// TIA Portal V17 export
// export: Created 2023-05-07T12:08:10.5778638Z, ExportSetting WithDefaults, DisplayName Totally Integrated Automation Portal, DisplayVersion V17, DisplayName TIA Portal Openness, DisplayVersion V17, DisplayName TIA Portal Version Control Interface, DisplayVersion V17, DisplayName TIA Portal Test Suite Advanced, DisplayVersion V17, DisplayName STEP 7 Professional, DisplayVersion V17, DisplayName SIMATIC Energy Suite, DisplayVersion V17, DisplayName STEP 7 Safety, DisplayVersion V17, DisplayName WinCC Professional, DisplayVersion V17
ORGANIZATION_BLOCK "Main"   // OB1, LAD, ProgramCycle
TITLE = "Main Program Sweep (Cycle)"
{ S7_Optimized_Access := 'TRUE' }
VERSION : 0.1
// stored: AutoNumber true, IsIECCheckEnabled false, SetENOAutomatically false
   VAR_INPUT
      Initial_Call : Bool;   // Initial call of this OB
      Remanence : Bool;   // =True, if remanent data are available
   END_VAR
BEGIN

REGION Network 1: Call: MHJ-PLC-Lab-Function-S71500
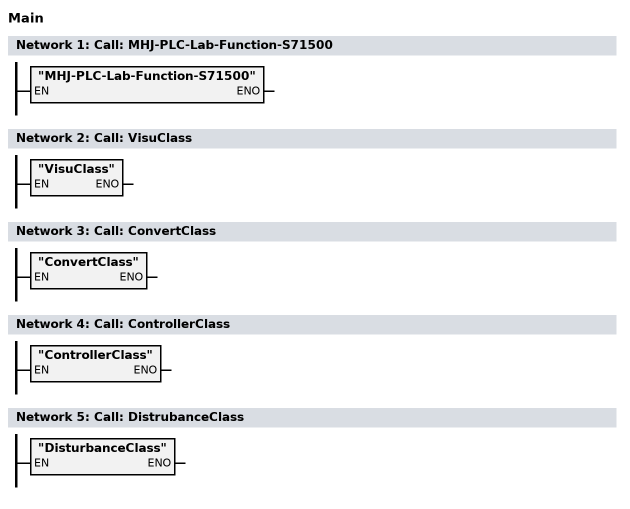
   RUNG wire#powerrail
      "MHJ-PLC-Lab-Function-S71500"()
   END_RUNG
   // the same network as SCL:
   "MHJ-PLC-Lab-Function-S71500"();
END_REGION

REGION Network 2: Call: VisuClass
   RUNG wire#powerrail
      "VisuClass"()
   END_RUNG
   // the same network as SCL:
   "VisuClass"();
END_REGION

REGION Network 3: Call: ConvertClass
   RUNG wire#powerrail
      "ConvertClass"()
   END_RUNG
   // the same network as SCL:
   "ConvertClass"();
END_REGION

REGION Network 4: Call: ControllerClass
   RUNG wire#powerrail
      "ControllerClass"()
   END_RUNG
   // the same network as SCL:
   "ControllerClass"();
END_REGION

REGION Network 5: Call: DistrubanceClass
   RUNG wire#powerrail
      "DisturbanceClass"()
   END_RUNG
   // the same network as SCL:
   "DisturbanceClass"();
END_REGION
END_ORGANIZATION_BLOCK
